PROGRAM MAIN
VAR
	comm			: FB_Comm_MQTT_Influx;
	RoofControl		: FB_RoofControl(comm := comm);
	
	// state
	closed			: BOOL;
	opened			: BOOL;
	stopped			: BOOL;
	opening			: BOOL;
	closing			: BOOL;
	error			: BOOL;
END_VAR

RoofControl(
	min_speed			:= 10000,
	max_speed 			:= 30000, 
	acceleration 		:= 150,
	max_position_1 		:= 200,
	max_position_2		:= 200,
	max_position_diff	:= 2,
	limit_slowdown		:= 5
);

comm(	
	sHostName		:= '10.129.129.76',
    nHostPort   	:= 1883,
    nKeepAlive  	:= 60,
	sTopicSub   	:= 'MONETN',
	sTopicLog		:= 'MONETN/Log',
	sTopicPublish	:= 'MONETN/Telemetry'
);


// state
closed 	:= RoofControl.State = E_RoofState.closed;
opened 	:= RoofControl.State = E_RoofState.opened;
stopped := RoofControl.State = E_RoofState.stopped;
opening := RoofControl.State = E_RoofState.opening;
closing := RoofControl.State = E_RoofState.closing;
error 	:= RoofControl.State = E_RoofState.error;

END_PROGRAM

(* stored: Version 1.1.0.1, ProductVersion 3.1.4024.15
   POU MAIN: Id {c6ad4756-c196-4e89-b031-015370ff4b7e}, SpecialFunc None *)
